(* CoDeSys 2.3.9.37 project: Cap6_4.pro *)
(* Libraries: Standard.lib 4.10.05 12:14:46 *)

(* POU PLC_PRG, LD *)
PROGRAM PLC_PRG
VAR
    (* Entradas *)
	A: BOOL;
	B: BOOL;
    (*Salidas *)
   	S1: BOOL;
      S2: BOOL;
    (*Instancias*)
 	MiTempo: TON;

END_VAR
VAR (* helpers for the ST form of the networks *)
	_p1 : BOOL;
END_VAR
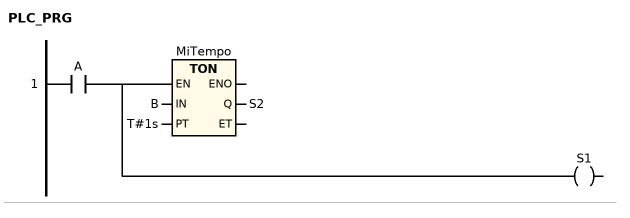
_LD_ (* Ladder Diagram *)
NETWORK 1
	[A] --- (S1)
		EN --- MiTempo:TON(IN: B, PT: T#1s) => S2
_END_LD_
(* the same logic as Structured Text *)
(* Network 1 *)
_p1 := A;
IF _p1 THEN
	MiTempo(IN := B, PT := T#1s);
	S2 := MiTempo.Q;
END_IF;
S1 := _p1;
END_PROGRAM

(* Visualisation Visu
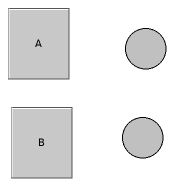
button at (41,30)-(102,101): text "A"; toggles PLC_PRG.A
ellipse at (158,50)-(199,91): alarm colour if PLC_PRG.S1
button at (44,129)-(105,200): text "B"; toggles PLC_PRG.B
ellipse at (155,139)-(196,180): alarm colour if PLC_PRG.S2
2 elements of other kinds (tables, trends, ...) not read
*)
